{attribute 'GeneratedUsingTerminal: EL3142--0000'}
{attribute addProperty BoxType "EL3142--0000"}
{attribute addProperty Id "Channel_1AT %I*Channel_7539AA333Channel_2AT %I*Channel_7539AA333WcStateAT %I*WcState_9091E0EB2InfoDataAT %I*InfoData_32EB74EA10"}
{attribute addProperty CRC "2161773851"}
{attribute addProperty Size "18"}
TYPE EL3142_80DA0D1B :
STRUCT
	{attribute addProperty Name "Channel_1"}
	Channel_1 : Channel_7539AA33;
	{attribute addProperty Name "Channel_2"}
	Channel_2 : Channel_7539AA33;
	{attribute addProperty Name "WcState"}
	WcState : WcState_9091E0EB;
	{attribute addProperty Name "InfoData"}
	InfoData : InfoData_32EB74EA;
END_STRUCT
END_TYPE

(* stored: Version 1.2.0.0, ProductVersion 3.1.4024.9
   DUT EL3142_80DA0D1B: Id {8800f746-e297-41f4-a1a2-a313a86aeeb1} *)
